// TIA Portal V17 export
// export: Created 2022-07-04T13:04:15.0491979Z, ExportSetting WithDefaults, DisplayName Totally Integrated Automation Portal, DisplayVersion V17, DisplayName TIA Portal Openness, DisplayVersion V17, DisplayName TIA Portal Version Control Interface, DisplayVersion V17, DisplayName STEP 7 Professional, DisplayVersion V17, DisplayName STEP 7 Safety, DisplayVersion V17, DisplayName WinCC Advanced, DisplayVersion V17
VAR_GLOBAL   // PLC tag table "Default tag table"
   opcUaConnect AT %M100.0 : Bool;
   opcUaRead AT %M100.1 : Bool;
   opcUaWrite AT %M100.2 : Bool;
   opcUaMethodCall AT %M100.3 : Bool;
   methodHdlIndex AT %MB0 : SInt;
END_VAR
VAR_GLOBAL CONSTANT   // user constants
   READ_LIST_COUNT : UInt := 3;
   WRITE_LIST_COUNT : UInt := 2;
   METHOD_LIST_COUNT : UInt := 1;
   NAMESPACE_COUNT : UInt := 1;
END_VAR
